(* IEC 61131-3 sources: Lasal/CPU_5344_V01/Class/EditString, 1 file *)

(* ---- EditString.st ---- *)
(*!
<Class
	Name               = "EditString"
	Revision           = "0.0"
	RealtimeTask       = "false"
	CyclicTask         = "false"
	BackgroundTask     = "false"
	Sigmatek           = "false"
	OSInterface        = "false"
	HighPriority       = "false"
	Automatic          = "false"
	UpdateMode         = "Prescan"
	SharedCommandTable = "true"
	Objectsize         = "(300,120)">
	<Channels>
		<Server Name="NewData" Visualized="false" Initialize="false" WriteProtected="false" Retentive="false"/>
	</Channels>
	<Network Name="EditString">
		<!-- List of Components in this network -->
		<Components>
			<Object
				Name       = "_base"
				Class      = "StringDll"
				Position   = "(241,120)"
				Visualized = "false">
				<Channels>
					<Server Name="Data"/>
					<Server Name="Handle"/>
				</Channels>
			</Object>
		</Components>
		<Comments>
		</Comments>
		<!-- List of Connections in this network -->
		<Connections>
			<Connection Source="this.Data" Destination="_base.Data" Vertices="(713,210),(541,210),"/>
			<Connection Source="this.Handle" Destination="_base.Handle" Vertices="(713,270),(541,270),"/>
		</Connections>
		<!-- Headerfiles -->
		<Options>
		</Options>
	</Network>
</Class>
*)
#pragma using StringDll

EditString : CLASS
: StringDll
  //Servers:
	NewData 	: SvrCh_DINT;
  //Clients:
  //Variables:
  //Functions:
				//! <Function Comment=" The function doesn&apos;t provide default functionality&#13;&#10; Please overwrite it for derived classes.&#13;&#10; Die Funktion stellt keine Standard-Implementierung dar. Sie muß für abgeleitete&#13;&#10; Klassen überschrieben werden.&#13;&#10;[&gt;udOff] Offset innerhalb des internen Datenpuffers, auf den die Daten kopiert werden sollen&#13;&#10;" Name="WriteDataOff"/>
	FUNCTION VIRTUAL GLOBAL WriteDataOff
		VAR_INPUT
			udLen 	: UDINT;			//! <Variable Comment="length of initialization data in bytes" Name="WriteDataOff.udLen"/>
			udOff 	: UDINT;			//! <Variable Comment=" offset where data should be copied to" Name="WriteDataOff.udOff"/>
			pData 	: ^USINT;
		END_VAR;
  //Tables:
	FUNCTION @STD
		VAR_OUTPUT
			ret_code	: CONFSTATES;
		END_VAR;
	FUNCTION GLOBAL TAB @CT_;
END_CLASS;

FUNCTION VIRTUAL GLOBAL EditString::WriteDataOff
	VAR_INPUT
		udLen 	: UDINT;
		udOff 	: UDINT;
		pData 	: ^USINT;
	END_VAR

  StringDll::WriteDataOff(udLen, udOff, pData);
  NewData += 1;

END_FUNCTION
